DATA_BLOCK "ST10_WarningDB"
{ S7_Optimized_Access := 'FALSE' }
VERSION : 0.1
// ATTRIBUTES
// AUTO_NUMBER = False
// BLOCK_NUMBER = 1068
// END_ATTRIBUTES
   STRUCT
      Global : Struct
         "1" : Struct
            PartLack1 : Bool;
            PartLack2 : Bool;
            PartLack3 : Bool;
            PartLack4 : Bool;
            PartLack5 : Bool;
            PartLack6 : Bool;
            PartLack7 : Bool;
            PartLack8 : Bool;
         END_STRUCT;
         "2" : Array[0..15] of Bool;
         "3" : Struct
            PartNoProperPosition1 : Bool;
            PartNoProperPosition2 : Bool;
            PartNoProperPosition3 : Bool;
            PartNoProperPosition4 : Bool;
            PartNoProperPosition5 : Bool;
            PartNoProperPosition6 : Bool;
            PartNoProperPosition7 : Bool;
            PartNoProperPosition8 : Bool;
         END_STRUCT;
         "4" : Array[0..15] of Bool;
         "5" : Struct
            ChangoverDataInvalide : Bool;
            PartDateInvalide : Bool;
            StationInHPToStart : Bool;
            lastStationPartNok : Bool;
         END_STRUCT;
         "6" : Array[0..15] of Bool;
         "7" : Array[0..15] of Bool;
         "8" : Array[0..15] of Bool;
         "9" : Array[0..15] of Bool;
         "10" : Array[0..15] of Bool;
      END_STRUCT;
      IndexTable : Array[1..2, 0..15] of Bool;
      Serve : Array[1..2, 0..15] of Bool;
      Servepress : Array[1..2, 0..15] of Bool;
      "3AxisServoInterpolation" : Array[1..2, 0..15] of Bool;
      LaserWelding : Array[1..2, 0..15] of Bool;
      LaserMarking : Array[1..2, 0..15] of Bool;
      Printer : Array[1..2, 0..15] of Bool;
      Marking : Array[1..2, 0..15] of Bool;
      Labelling : Array[1..2, 0..15] of Bool;
      Dispensing : Array[1..2, 0..15] of Bool;
      GreasingSystem : Array[1..2, 0..15] of Bool;
      HotWindSystem : Array[1..2, 0..15] of Bool;
      HighFrequencyHeating : Array[1..2, 0..15] of Bool;
      Degaussing : Array[1..2, 0..15] of Bool;
      BowlFeeder : Array[1..2, 0..15] of Bool;
      Riveter : Array[1..2, 0..15] of Bool;
      HydraulicSystem : Array[1..2, 0..15] of Bool;
      Robot : Array[1..2, 0..15] of Bool;
      Camera : Array[1..2, 0..15] of Bool;
      Scannner : Array[1..2, 0..15] of Bool;
      MeasureSensor : Array[1..2, 0..15] of Bool;
      Leakage : Array[1..2, 0..15] of Bool;
      TestPowerSupply : Array[1..2, 0..15] of Bool;
      HighVoltageTester : Array[1..2, 0..15] of Bool;
      EOLfinalInspection : Array[1..2, 0..15] of Bool;
      Screw : Array[1..2, 0..15] of Bool;
      "3AxisScrewEncoder" : Array[1..2, 0..15] of Bool;
      Heating : Array[1..2, 0..15] of Bool;
      PressurizedOilAirCylinder : Array[1..2, 0..15] of Bool;
      Moby : Array[1..2, 0..15] of Bool;
      IPC : Array[1..2, 0..15] of Bool;
      ValveIsland : Array[1..2, 0..15] of Bool;
      RFID : Array[1..2, 0..15] of Bool;
      RemoteIO : Array[1..2, 0..15] of Bool;
      DPSlaveStation : Array[1..2, 0..15] of Bool;
      MSCOMM : Array[1..2, 0..15] of Bool;
      Flowtester : Array[1..2, 0..15] of Bool;
      CurrentsTester : Array[1..2, 0..15] of Bool;
      VoltageTester : Array[1..2, 0..15] of Bool;
      InductanceTester : Array[1..2, 0..15] of Bool;
      ResistanceTester : Array[1..2, 0..15] of Bool;
      LCRTester : Array[1..2, 0..15] of Bool;
      PressureDisplacementMonitor : Array[1..2, 0..15] of Bool;
      UltrasonicWelding : Array[1..2, 0..15] of Bool;
      ElectricResistanceWelding : Array[1..2, 0..15] of Bool;
   END_STRUCT;


BEGIN

END_DATA_BLOCK

